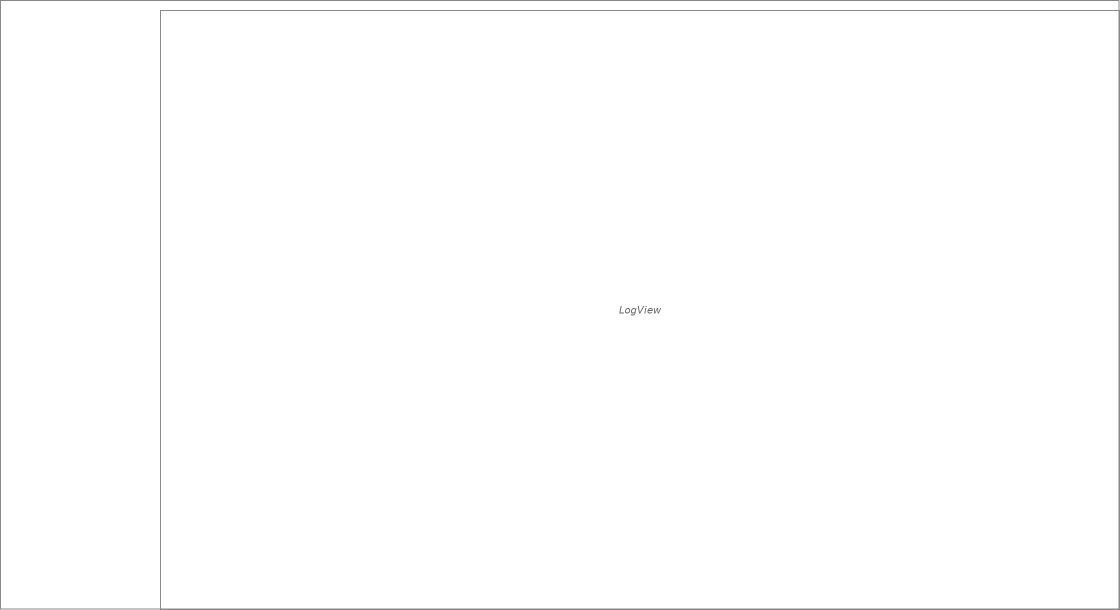
VISUALIZATION Log_  // 1120x610
    Frame (160,10 960x600)
        shows LogView(fbLogView := GVL_HMI.fbHMIControl.fbLogView)
END_VISUALIZATION

(* stored: Version 1.1.0.1, ProductVersion 3.1.4024.11
   Visu Log_: Id {9d1d492b-4ead-40bc-8482-c9349fd92015} *)
